{attribute addProperty BoxType "AT2050-5500-0018"}
{attribute addProperty Id "FB_InputsAT %I*FB_Inputs_A6E87AE0528660FB_OutputsAT %Q*FB_Outputs_734938A41620WcStateAT %I*WcState_F855686C1620InfoDataAT %I*InfoData_7231B2DD80100"}
{attribute addProperty CRC "609416669"}
{attribute addProperty SizeInBites "640"}
{attribute addProperty SizeInBytes "80"}
TYPE AT2050_3DCFC8D0 :
STRUCT
	{attribute addProperty Name "FB_Inputs"}
	FB_Inputs : FB_Inputs_A6E87AE0;
	{attribute addProperty Name "FB_Outputs"}
	FB_Outputs : FB_Outputs_734938A4;
	{attribute addProperty Name "WcState"}
	WcState : WcState_F855686C;
	{attribute addProperty Name "InfoData"}
	InfoData : InfoData_7231B2DD;
END_STRUCT
END_TYPE

(* stored: Version 1.2.0.0, ProductVersion 3.1.4024.9
   DUT AT2050_3DCFC8D0: Id {d3cff985-11f9-4dac-9fca-a9d132030f6f} *)
